{attribute 'TcGenerated'}
// This function has been automatically generated from the project information.
VAR_GLOBAL CONSTANT
    {attribute 'const_non_replaced'}
    {attribute 'linkalways'}
    stLibVersion_plc_kfe_rix_motion : ST_LibVersion := (iMajor := 1, iMinor := 0, iBuild := 1, iRevision := 0, sVersion := '1.0.1');
END_VAR

(* stored: Version 1.1.0.1, ProductVersion 3.1.4024.2
   GVL Global_Version: Id b2d22559-f359-41a9-8aad-d34621ada962 *)
